FUNCTION_BLOCK FB_SignalHandlingDelay EXTENDS FB_SignalHandling
VAR_INPUT
	tDelay						:			TIME;				// Time to delay input signal
END_VAR
VAR_OUTPUT
END_VAR
VAR
	bStartProcessingDelay		:			BOOL;				// Bit for releasing processing of input delay
	fbTimerDelay				:			TON;				// Timer to control processing delay of input signal
END_VAR

METHOD SetOutput
	IF bInputSignal AND bEnableInputLocal THEN
		bStartProcessingDelay 	:= 		TRUE;
	END_IF

	IF	bStartProcessingDelay THEN
		fbTimerDelay(	IN		:=		TRUE,
						PT		:=		tDelay);
	ELSE
		fbTimerDelay(	IN		:=		FALSE);
	END_IF

	IF fbTimerDelay.Q THEN
		bStartProcessingDelay	:=		FALSE;

		fbTimerDelay(	IN		:=		FALSE);	 
		
		bOutputSignal			:=		TRUE;
	ELSE
		bOutputSignal			:=		FALSE;
	END_IF
END_METHOD

END_FUNCTION_BLOCK

(* stored: Version 1.1.0.1, ProductVersion 3.1.4024.15
   POU FB_SignalHandlingDelay: Id {06a2ad3f-9776-43e7-8e5a-9eb687aa8e24}, SpecialFunc None
   Method SetOutput: Id {56e929ac-4eee-47f6-839e-14434f37a3af} *)
